(* PLC project Unnamed, Desconocido Unnamed 1 *)
(* stored: creationDateTime 2026-03-01T14:16:40, modificationDateTime 2026-03-16T02:26:01 *)

FUNCTION_BLOCK functionBlock0
  VAR_INPUT
    In0 : BOOL := 0;
    In1 : BOOL := 0;
  END_VAR
  VAR_OUTPUT
    Out1 : BOOL := 0;
  END_VAR
  VAR
    Out2 : BOOL := 0;
  END_VAR

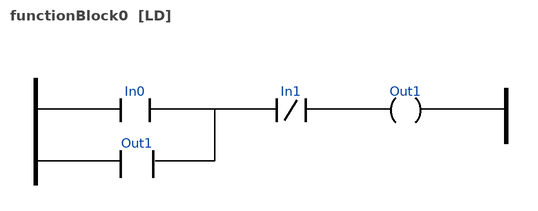
(* LD diagram, written out as Structured Text *)
Out1 := (In0 OR Out1) AND NOT In1;
END_FUNCTION_BLOCK

PROGRAM program0
  VAR
    functionBlock00 : functionBlock0;
  END_VAR
  VAR_INPUT
    Input1 : BOOL := 0;  (* leer con gpio_get_level(PIN_IN1) *)
    Input2 : BOOL := 0;  (* leer con gpio_get_level(PIN_IN2) *)
  END_VAR
  VAR_OUTPUT
    Output1 : BOOL := 0;  (* leer con gpio_set_level(PIN_OUT2) *)
    Output2 : BOOL := 0;  (* leer con gpio_set_level(PIN_OUT2) *)
  END_VAR
  VAR_INPUT
    Start : BOOL := 0;  (* leer con gpio_set_level(PIN_OUT2) *)
  END_VAR
  VAR_OUTPUT
    Done : BOOL := 0;  (* leer con gpio_set_level(PIN_OUT2) *)
    Busy : BOOL := 0;  (* leer con gpio_set_level(PIN_OUT2) *)
    Error : BOOL := 0;  (* leer con gpio_set_level(PIN_OUT2) *)
  END_VAR
  VAR_INPUT
    TargetPos : LREAL := 10.1;  (* leer con gpio_set_level(PIN_OUT2) *)
    Speed : LREAL := 1.1;  (* leer con gpio_set_level(PIN_OUT2) *)
  END_VAR
  VAR
    functionBlock01 : functionBlock0;
  END_VAR

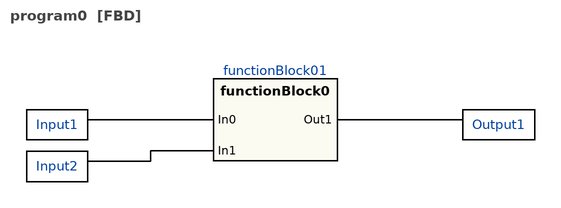
(* FBD diagram, written out as Structured Text *)
functionBlock01(In0 := Input1, In1 := Input2);
Output1 := functionBlock01.Out1;
END_PROGRAM

CONFIGURATION config
  RESOURCE resource1 ON PLC
    TASK task0(INTERVAL := T#20ms, PRIORITY := 0);
    PROGRAM instance0 WITH task0 : program0;
  END_RESOURCE
END_CONFIGURATION
